INTERFACE I_ListBase

{attribute 'OPC.UA.DA.Property' := '1'}
{attribute 'monitoring' := 'call'}
PROPERTY public P_Length : DINT
GET
END_GET
END_PROPERTY

METHOD PUBLIC M_Clear : BOOL
END_METHOD

END_INTERFACE

(* stored: Version 1.1.0.1
   Itf I_ListBase: Id {a3cd9153-0c75-00d3-05d8-20fe19f8ccb0}
   Property P_Length: Id {49615258-7cc8-4370-999e-56e1024f4c79}
   Get Get: Id {ec48dc05-e74e-4cfe-acf2-317ea9ff6055}
   Method M_Clear: Id {bec35183-59fd-4e05-8c88-04323521ec68} *)
